TYPE ST_MOVER_OFFSETS :
STRUCT
  // static position offsets in stations
  PositionOffset      : ARRAY[1..MAX_STATION] OF T_NEST_OFFSET; // added to PosStop[] in XtsStation
END_STRUCT
END_TYPE

(* stored: Version 1.1.0.1, ProductVersion 3.1.4026.18
   DUT ST_MOVER_OFFSETS: Id {c7cde426-a6c1-447f-aed7-b3c881333fc8} *)
